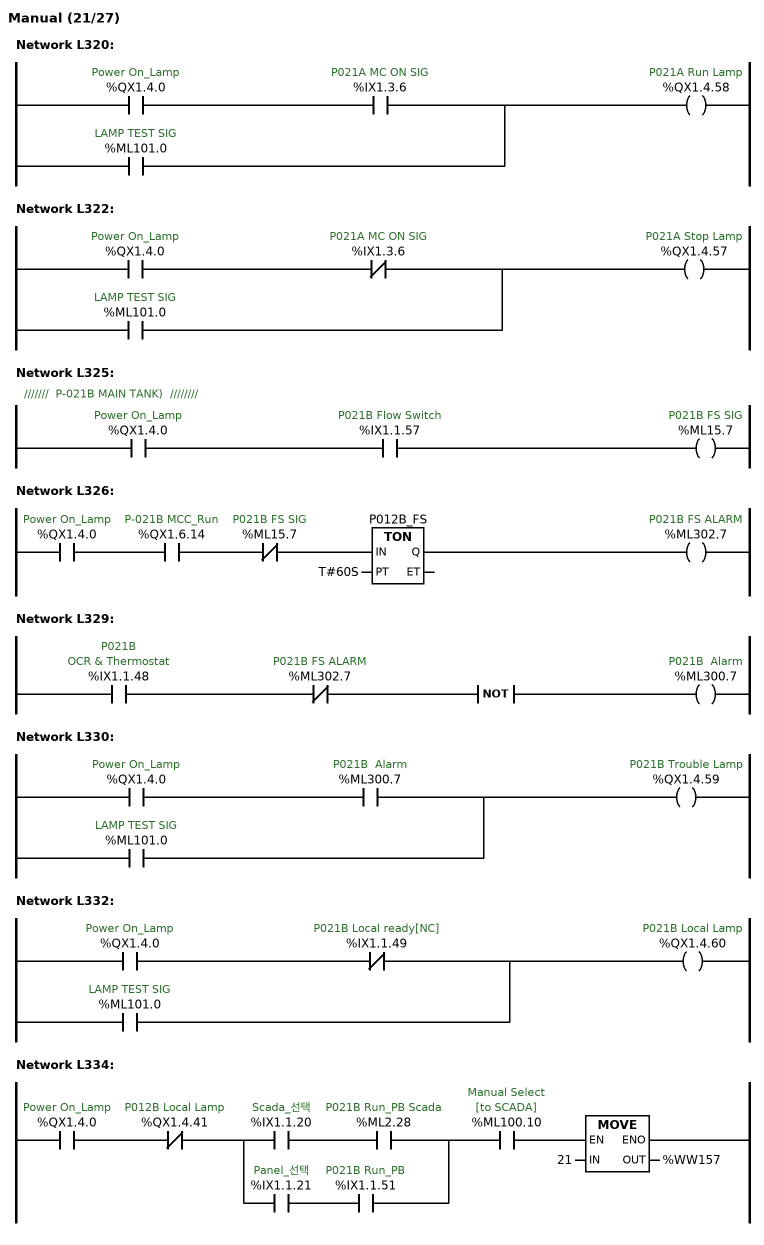
(* [picture p24: Manual rungs L320-L334] *)
(* Rung L320 *)
%QX1.4.58 := (%QX1.4.0 AND %IX1.3.6) OR %ML101.0;
(* Rung L322 *)
%QX1.4.57 := (%QX1.4.0 AND NOT %IX1.3.6) OR %ML101.0;
(* ///////  P-021B MAIN TANK)  //////// *)
(* Rung L325 *)
%ML15.7 := %QX1.4.0 AND %IX1.1.57;
(* Rung L326 *)
P012B_FS(IN := %QX1.4.0 AND %QX1.6.14 AND NOT %ML15.7, PT := T#60S);
%ML302.7 := P012B_FS.Q;
(* Rung L329 *)
%ML300.7 := NOT (%IX1.1.48 AND NOT %ML302.7);
(* Rung L330 *)
%QX1.4.59 := (%QX1.4.0 AND %ML300.7) OR %ML101.0;
(* Rung L332 *)
%QX1.4.60 := (%QX1.4.0 AND NOT %IX1.1.49) OR %ML101.0;
(* Rung L334 *)
IF %QX1.4.0 AND NOT %QX1.4.41 AND ((%IX1.1.20 AND %ML2.28) OR (%IX1.1.21 AND %IX1.1.51)) AND %ML100.10 THEN
    %WW157 := 21;
END_IF;

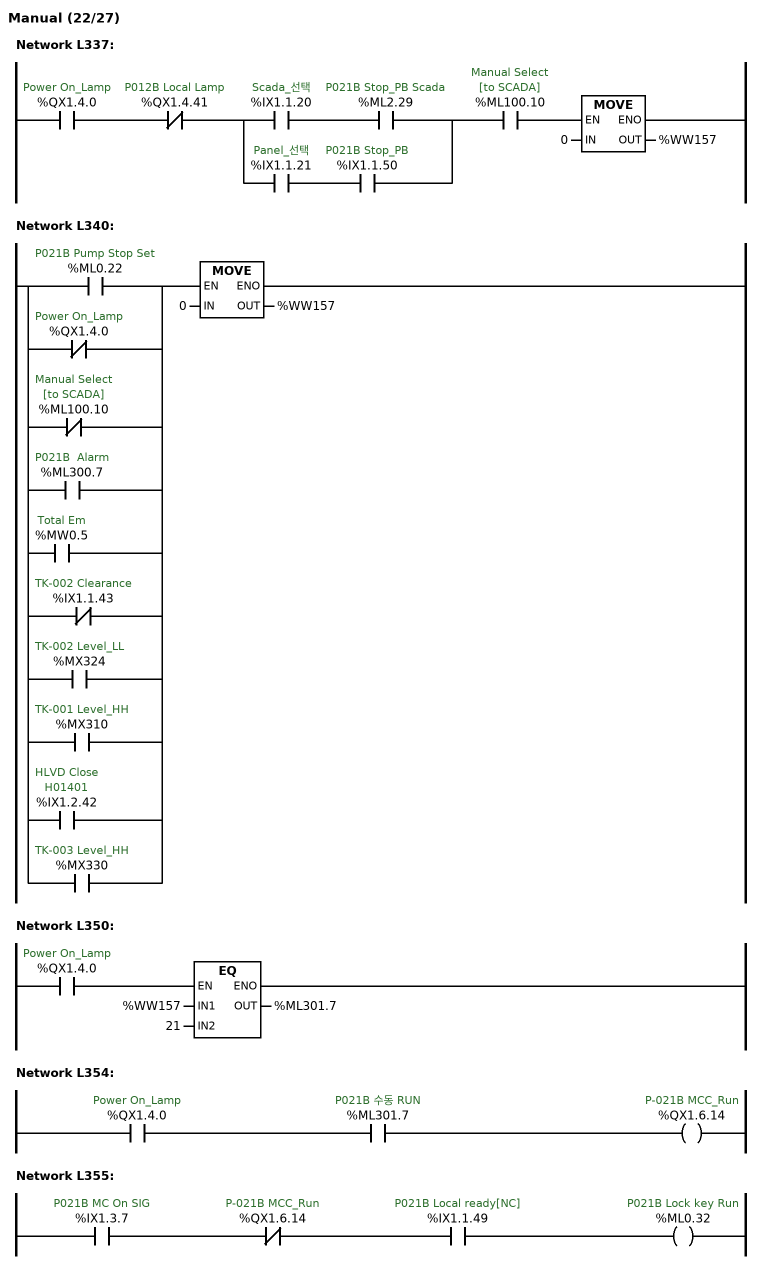
(* Rung L337 *)
IF %QX1.4.0 AND NOT %QX1.4.41 AND ((%IX1.1.20 AND %ML2.29) OR (%IX1.1.21 AND %IX1.1.50)) AND %ML100.10 THEN
    %WW157 := 0;
END_IF;
(* Rung L340 *)
IF %ML0.22 OR NOT %QX1.4.0 OR NOT %ML100.10 OR %ML300.7 OR %MW0.5 OR NOT %IX1.1.43 OR %MX324 OR %MX310 OR %IX1.2.42 OR %MX330 THEN
    %WW157 := 0;
END_IF;
(* Rung L350 *)
IF %QX1.4.0 THEN %ML301.7 := %WW157 = 21; END_IF;
(* Rung L354 *)
%QX1.6.14 := %QX1.4.0 AND %ML301.7;
(* Rung L355 *)
%ML0.32 := %IX1.3.7 AND NOT %QX1.6.14 AND %IX1.1.49;

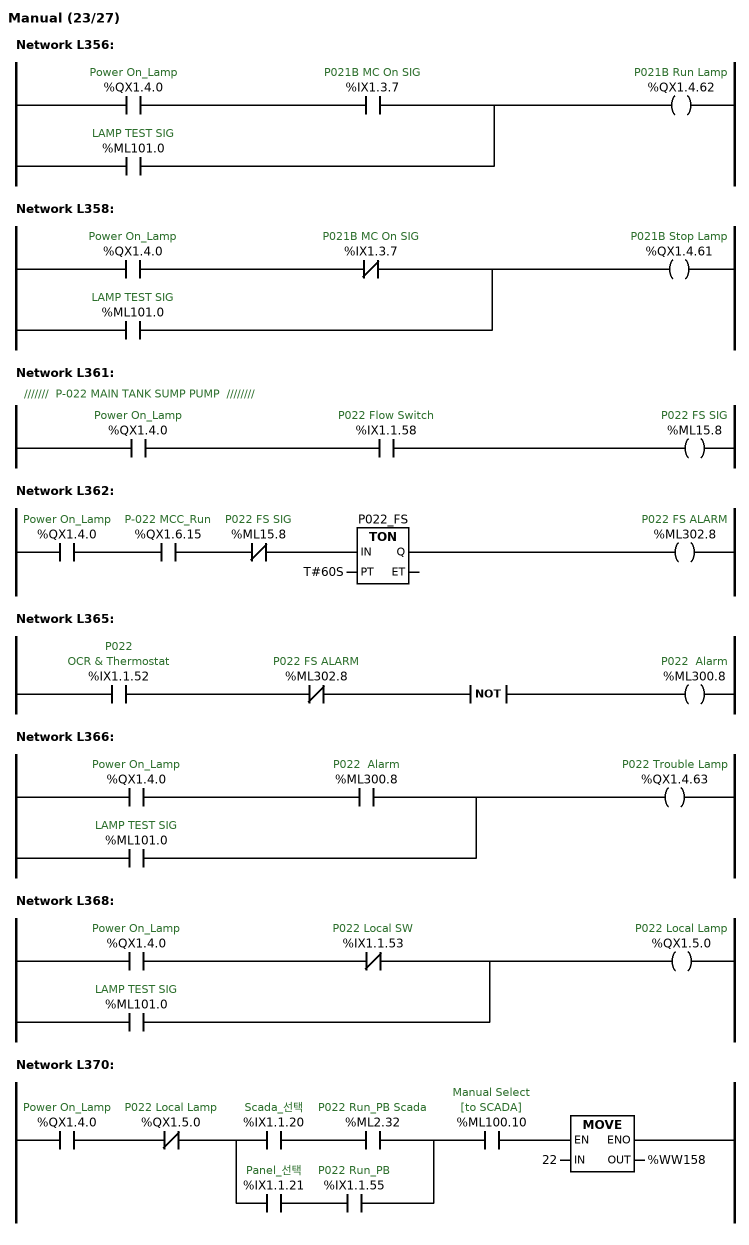
(* Rung L356 *)
%QX1.4.62 := (%QX1.4.0 AND %IX1.3.7) OR %ML101.0;
(* Rung L358 *)
%QX1.4.61 := (%QX1.4.0 AND NOT %IX1.3.7) OR %ML101.0;
(* ///////  P-022 MAIN TANK SUMP PUMP  //////// *)
(* Rung L361 *)
%ML15.8 := %QX1.4.0 AND %IX1.1.58;
(* Rung L362 *)
P022_FS(IN := %QX1.4.0 AND %QX1.6.15 AND NOT %ML15.8, PT := T#60S);
%ML302.8 := P022_FS.Q;
(* Rung L365 *)
%ML300.8 := NOT (%IX1.1.52 AND NOT %ML302.8);
(* Rung L366 *)
%QX1.4.63 := (%QX1.4.0 AND %ML300.8) OR %ML101.0;
(* Rung L368 *)
%QX1.5.0 := (%QX1.4.0 AND NOT %IX1.1.53) OR %ML101.0;
(* Rung L370 *)
IF %QX1.4.0 AND NOT %QX1.5.0 AND ((%IX1.1.20 AND %ML2.32) OR (%IX1.1.21 AND %IX1.1.55)) AND %ML100.10 THEN
    %WW158 := 22;
END_IF;

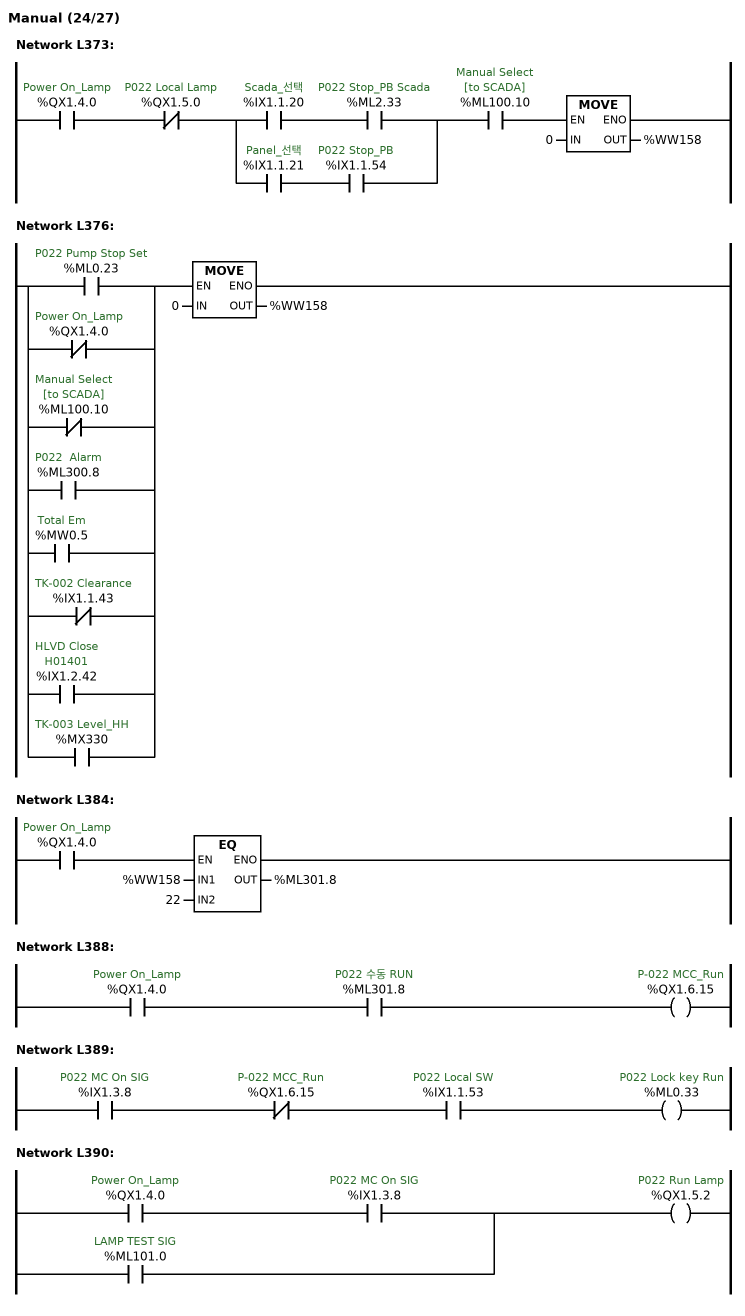
(* Rung L373 *)
IF %QX1.4.0 AND NOT %QX1.5.0 AND ((%IX1.1.20 AND %ML2.33) OR (%IX1.1.21 AND %IX1.1.54)) AND %ML100.10 THEN
    %WW158 := 0;
END_IF;
(* Rung L376 *)
IF %ML0.23 OR NOT %QX1.4.0 OR NOT %ML100.10 OR %ML300.8 OR %MW0.5 OR NOT %IX1.1.43 OR %IX1.2.42 OR %MX330 THEN
    %WW158 := 0;
END_IF;
(* Rung L384 *)
IF %QX1.4.0 THEN %ML301.8 := %WW158 = 22; END_IF;
(* Rung L388 *)
%QX1.6.15 := %QX1.4.0 AND %ML301.8;
(* Rung L389 *)
%ML0.33 := %IX1.3.8 AND NOT %QX1.6.15 AND %IX1.1.53;
(* Rung L390 *)
%QX1.5.2 := (%QX1.4.0 AND %IX1.3.8) OR %ML101.0;

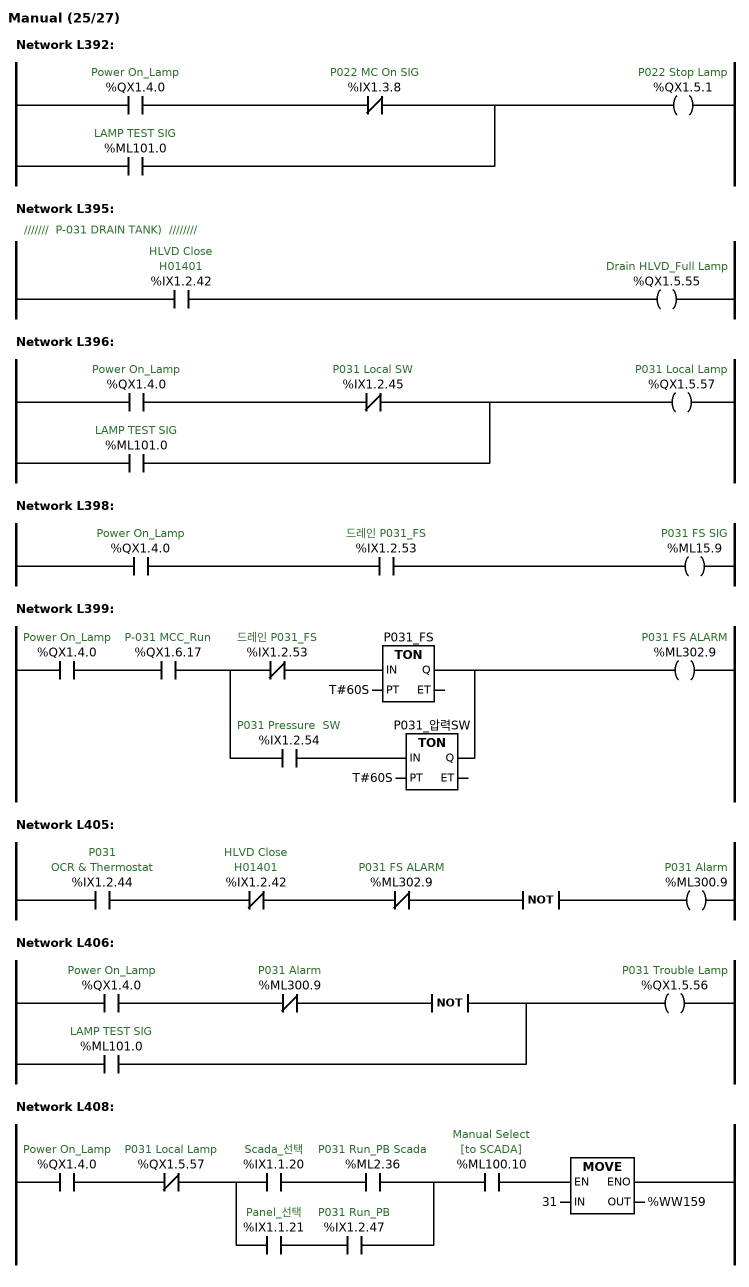
(* Rung L392 *)
%QX1.5.1 := (%QX1.4.0 AND NOT %IX1.3.8) OR %ML101.0;
(* ///////  P-031 DRAIN TANK)  //////// *)
(* Rung L395 *)
%QX1.5.55 := %IX1.2.42;
(* Rung L396 *)
%QX1.5.57 := (%QX1.4.0 AND NOT %IX1.2.45) OR %ML101.0;
(* Rung L398 *)
%ML15.9 := %QX1.4.0 AND %IX1.2.53;
(* Rung L399 *)
P031_FS(IN := %QX1.4.0 AND %QX1.6.17 AND NOT %IX1.2.53, PT := T#60S);
P031_압력SW(IN := %QX1.4.0 AND %QX1.6.17 AND %IX1.2.54, PT := T#60S);
%ML302.9 := P031_FS.Q OR P031_압력SW.Q;
(* Rung L405 *)
%ML300.9 := NOT (%IX1.2.44 AND NOT %IX1.2.42 AND NOT %ML302.9);
(* Rung L406 *)
%QX1.5.56 := NOT (%QX1.4.0 AND NOT %ML300.9) OR %ML101.0;
(* Rung L408 *)
IF %QX1.4.0 AND NOT %QX1.5.57 AND ((%IX1.1.20 AND %ML2.36) OR (%IX1.1.21 AND %IX1.2.47)) AND %ML100.10 THEN
    %WW159 := 31;
END_IF;

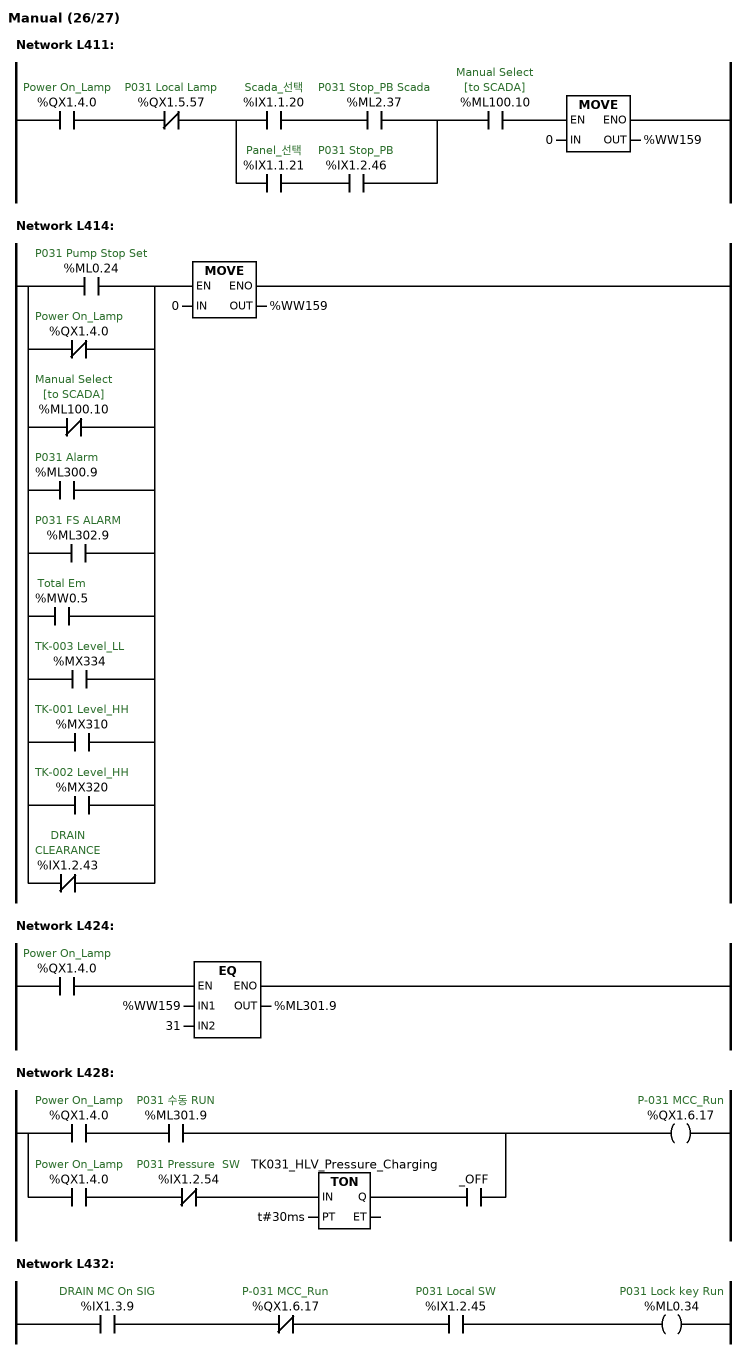
(* Rung L411 *)
IF %QX1.4.0 AND NOT %QX1.5.57 AND ((%IX1.1.20 AND %ML2.37) OR (%IX1.1.21 AND %IX1.2.46)) AND %ML100.10 THEN
    %WW159 := 0;
END_IF;
(* Rung L414 *)
IF %ML0.24 OR NOT %QX1.4.0 OR NOT %ML100.10 OR %ML300.9 OR %ML302.9 OR %MW0.5 OR %MX334 OR %MX310 OR %MX320 OR NOT %IX1.2.43 THEN
    %WW159 := 0;
END_IF;
(* Rung L424 *)
IF %QX1.4.0 THEN %ML301.9 := %WW159 = 31; END_IF;
(* Rung L428 *)
TK031_HLV_Pressure_Charging(IN := %QX1.4.0 AND NOT %IX1.2.54, PT := t#30ms);
%QX1.6.17 := (%QX1.4.0 AND %ML301.9) OR (TK031_HLV_Pressure_Charging.Q AND _OFF);
(* Rung L432 *)
%ML0.34 := %IX1.3.9 AND NOT %QX1.6.17 AND %IX1.2.45;

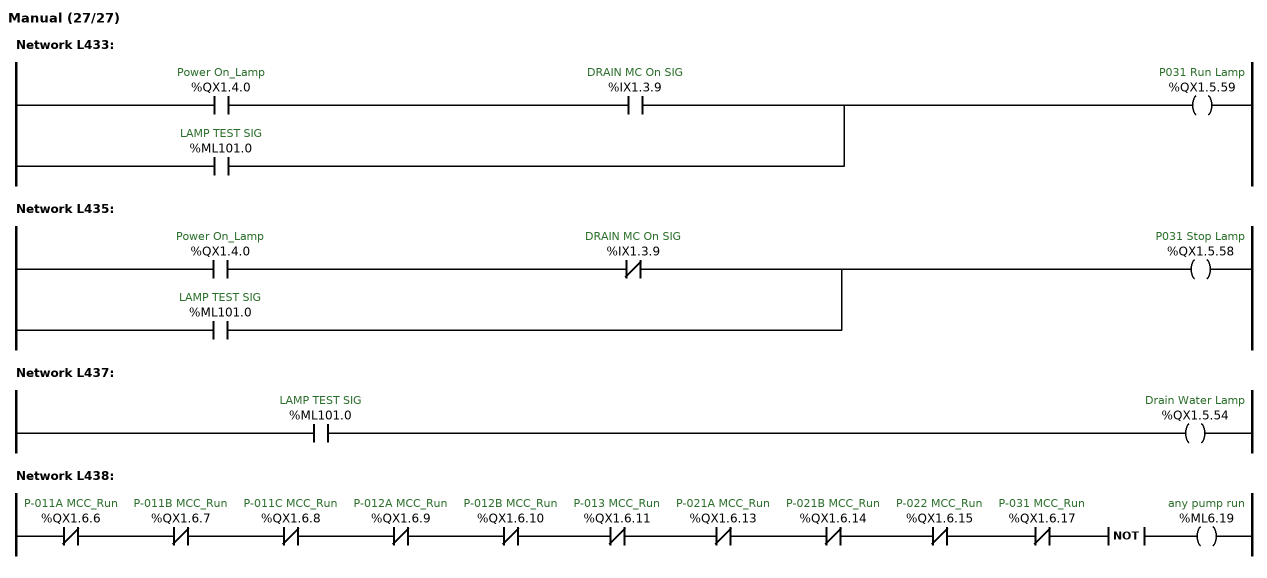
(* Rung L433 *)
%QX1.5.59 := (%QX1.4.0 AND %IX1.3.9) OR %ML101.0;
(* Rung L435 *)
%QX1.5.58 := (%QX1.4.0 AND NOT %IX1.3.9) OR %ML101.0;
(* Rung L437 *)
%QX1.5.54 := %ML101.0;
(* Rung L438 *)
%ML6.19 := NOT (NOT %QX1.6.6 AND NOT %QX1.6.7 AND NOT %QX1.6.8 AND NOT %QX1.6.9 AND NOT %QX1.6.10 AND NOT %QX1.6.11 AND NOT %QX1.6.13 AND NOT %QX1.6.14 AND NOT %QX1.6.15 AND NOT %QX1.6.17);
END_PROGRAM

PROGRAM Automatic (* task: 스캔 프로그램 *)
VAR
    AUTO_S_FS : TON;
END_VAR

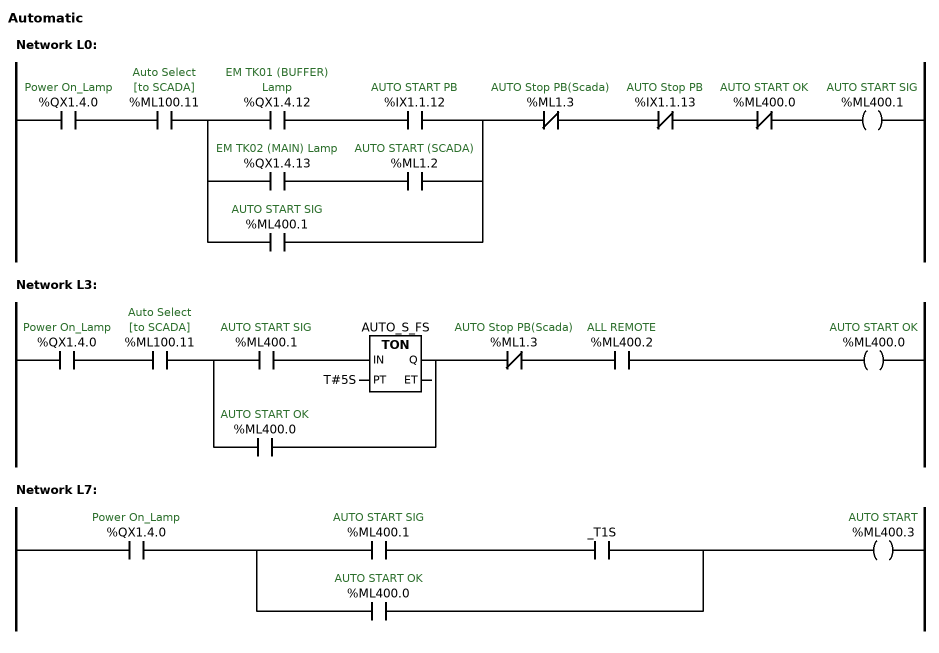
(* Rung L0 *)
%ML400.1 := %QX1.4.0 AND %ML100.11 AND ((%QX1.4.12 AND %IX1.1.12) OR (%QX1.4.13 AND %ML1.2) OR %ML400.1) AND NOT %ML1.3 AND NOT %IX1.1.13 AND NOT %ML400.0;
(* Rung L3 *)
AUTO_S_FS(IN := %QX1.4.0 AND %ML100.11 AND %ML400.1, PT := T#5S);
%ML400.0 := (AUTO_S_FS.Q OR (%QX1.4.0 AND %ML100.11 AND %ML400.0)) AND NOT %ML1.3 AND %ML400.2;
(* Rung L7 *)
%ML400.3 := %QX1.4.0 AND ((%ML400.1 AND _T1S) OR %ML400.0);
END_PROGRAM

PROGRAM Analog (* task: 스캔 프로그램 *)
VAR_EXTERNAL
    _0100_CH0_ACT : BOOL; (* AT %UX1.0.16 *) (* 아날로그입력 모듈: 채널0 운전중 *)
    _0100_CH0_DATA : INT; (* AT %UW1.0.2 *) (* 아날로그입력 모듈: 채널0 변환값 *)
    _0100_CH0_IDD : BOOL; (* AT %UX1.0.160 *) (* 아날로그입력 모듈: 채널0 입력단선검출 *)
    _0100_CH1_ACT : BOOL; (* AT %UX1.0.17 *) (* 아날로그입력 모듈: 채널1 운전중 *)
    _0100_CH1_DATA : INT; (* AT %UW1.0.3 *) (* 아날로그입력 모듈: 채널1 변환값 *)
    _0100_CH1_IDD : BOOL; (* AT %UX1.0.161 *) (* 아날로그입력 모듈: 채널1 입력단선검출 *)
    _0100_CH2_ACT : BOOL; (* AT %UX1.0.18 *) (* 아날로그입력 모듈: 채널2 운전중 *)
    _0100_CH2_DATA : INT; (* AT %UW1.0.4 *) (* 아날로그입력 모듈: 채널2 변환값 *)
    _0100_CH2_IDD : BOOL; (* AT %UX1.0.162 *) (* 아날로그입력 모듈: 채널2 입력단선검출 *)
    _0100_CH3_ACT : BOOL; (* AT %UX1.0.19 *) (* 아날로그입력 모듈: 채널3 운전중 *)
    _0100_CH3_DATA : INT; (* AT %UW1.0.5 *) (* 아날로그입력 모듈: 채널3 변환값 *)
    _0100_CH3_IDD : BOOL; (* AT %UX1.0.163 *) (* 아날로그입력 모듈: 채널3 입력단선검출 *)
    _0100_CH4_ACT : BOOL; (* AT %UX1.0.20 *) (* 아날로그입력 모듈: 채널4 운전중 *)
    _0100_CH4_DATA : INT; (* AT %UW1.0.6 *) (* 아날로그입력 모듈: 채널4 변환값 *)
    _0100_CH4_IDD : BOOL; (* AT %UX1.0.164 *) (* 아날로그입력 모듈: 채널4 입력단선검출 *)
    _0100_CH5_ACT : BOOL; (* AT %UX1.0.21 *) (* 아날로그입력 모듈: 채널5 운전중 *)
    _0100_CH5_DATA : INT; (* AT %UW1.0.7 *) (* 아날로그입력 모듈: 채널5 변환값 *)
    _0100_CH5_IDD : BOOL; (* AT %UX1.0.165 *) (* 아날로그입력 모듈: 채널5 입력단선검출 *)
    _0100_CH6_ACT : BOOL; (* AT %UX1.0.22 *) (* 아날로그입력 모듈: 채널6 운전중 *)
    _0100_CH6_DATA : INT; (* AT %UW1.0.8 *) (* 아날로그입력 모듈: 채널6 변환값 *)
    _0100_CH6_IDD : BOOL; (* AT %UX1.0.166 *) (* 아날로그입력 모듈: 채널6 입력단선검출 *)
    _0100_CH7_ACT : BOOL; (* AT %UX1.0.23 *) (* 아날로그입력 모듈: 채널7 운전중 *)
    _0100_CH7_DATA : INT; (* AT %UW1.0.9 *) (* 아날로그입력 모듈: 채널7 변환값 *)
    _0100_CH7_IDD : BOOL; (* AT %UX1.0.167 *) (* 아날로그입력 모듈: 채널7 입력단선검출 *)
END_VAR
VAR
    _t1 : BOOL;
    _t2 : BOOL;
    _t3 : BOOL;
    _t4 : BOOL;
END_VAR

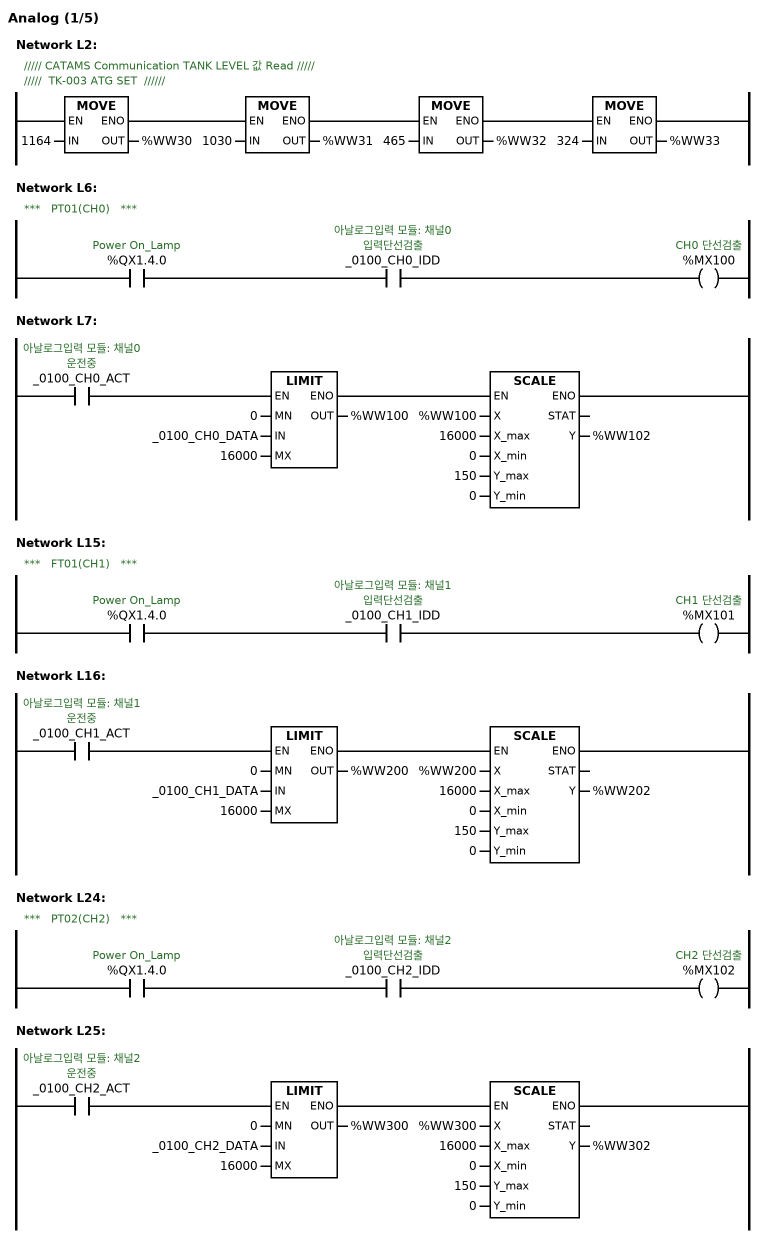
(* ///// CATAMS Communication TANK LEVEL 값 Read ///// *)
(* /////  TK-003 ATG SET  ////// *)
(* Rung L2 *)
%WW30 := 1164;
%WW31 := 1030;
%WW32 := 465;
%WW33 := 324;
(* ***   PT01(CH0)   *** *)
(* Rung L6 *)
%MX100 := %QX1.4.0 AND _0100_CH0_IDD;
(* Rung L7 *)
IF _0100_CH0_ACT THEN
    %WW100 := LIMIT(MN := 0, IN := _0100_CH0_DATA, MX := 16000);
    SCALE(X := %WW100, X_max := 16000, X_min := 0, Y_max := 150, Y_min := 0, Y => %WW102);
END_IF;
(* ***   FT01(CH1)   *** *)
(* Rung L15 *)
%MX101 := %QX1.4.0 AND _0100_CH1_IDD;
(* Rung L16 *)
IF _0100_CH1_ACT THEN
    %WW200 := LIMIT(MN := 0, IN := _0100_CH1_DATA, MX := 16000);
    SCALE(X := %WW200, X_max := 16000, X_min := 0, Y_max := 150, Y_min := 0, Y => %WW202);
END_IF;
(* ***   PT02(CH2)   *** *)
(* Rung L24 *)
%MX102 := %QX1.4.0 AND _0100_CH2_IDD;
(* Rung L25 *)
IF _0100_CH2_ACT THEN
    %WW300 := LIMIT(MN := 0, IN := _0100_CH2_DATA, MX := 16000);
    SCALE(X := %WW300, X_max := 16000, X_min := 0, Y_max := 150, Y_min := 0, Y => %WW302);
END_IF;

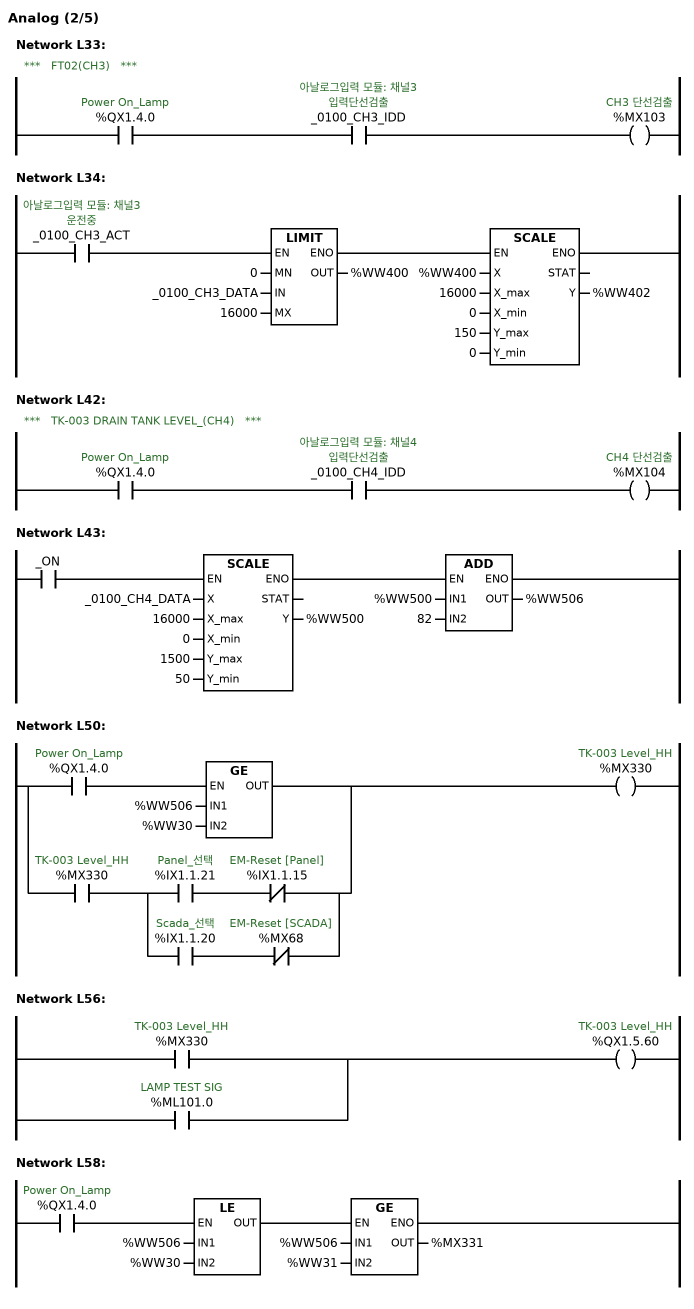
(* ***   FT02(CH3)   *** *)
(* Rung L33 *)
%MX103 := %QX1.4.0 AND _0100_CH3_IDD;
(* Rung L34 *)
IF _0100_CH3_ACT THEN
    %WW400 := LIMIT(MN := 0, IN := _0100_CH3_DATA, MX := 16000);
    SCALE(X := %WW400, X_max := 16000, X_min := 0, Y_max := 150, Y_min := 0, Y => %WW402);
END_IF;
(* ***   TK-003 DRAIN TANK LEVEL_(CH4)   *** *)
(* Rung L42 *)
%MX104 := %QX1.4.0 AND _0100_CH4_IDD;
(* Rung L43 *)
IF _ON THEN
    SCALE(X := _0100_CH4_DATA, X_max := 16000, X_min := 0, Y_max := 1500, Y_min := 50, Y => %WW500);
    %WW506 := %WW500 + 82;
END_IF;
(* Rung L50 *)
IF %QX1.4.0 THEN _t1 := %WW506 >= %WW30; END_IF;
%MX330 := _t1 OR (%MX330 AND ((%IX1.1.21 AND NOT %IX1.1.15) OR (%IX1.1.20 AND NOT %MX68)));
(* Rung L56 *)
%QX1.5.60 := %MX330 OR %ML101.0;
(* Rung L58 *)
IF %QX1.4.0 THEN _t2 := %WW506 <= %WW30; END_IF;
IF _t2 THEN %MX331 := %WW506 >= %WW31; END_IF;

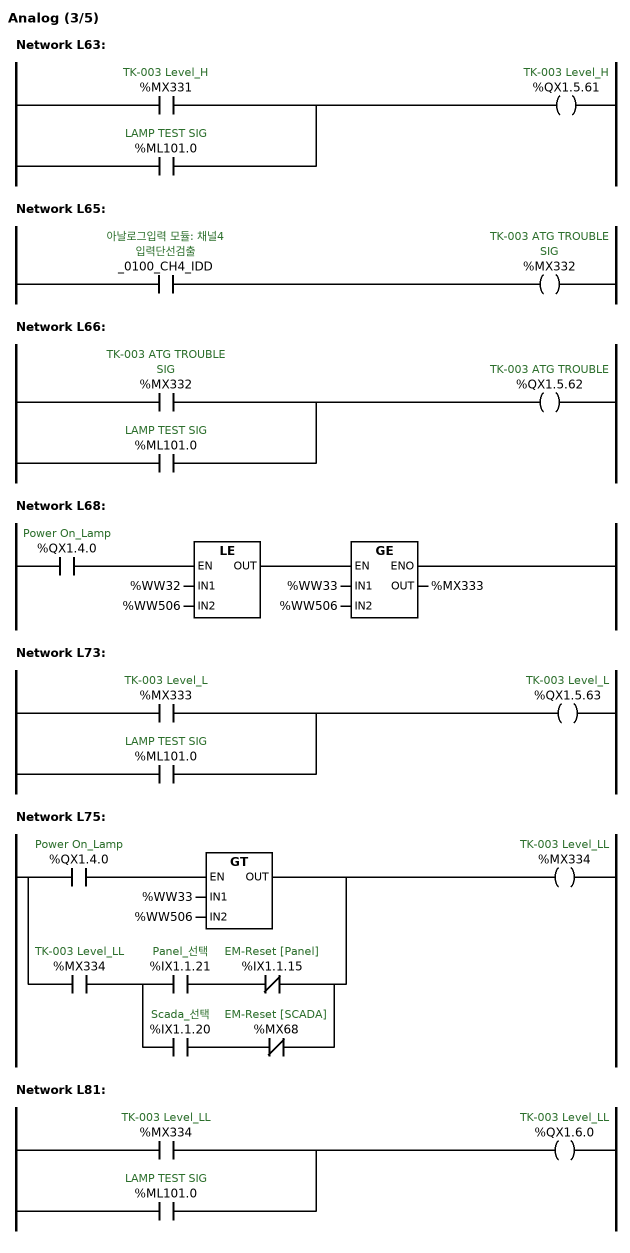
(* Rung L63 *)
%QX1.5.61 := %MX331 OR %ML101.0;
(* Rung L65 *)
%MX332 := _0100_CH4_IDD;
(* Rung L66 *)
%QX1.5.62 := %MX332 OR %ML101.0;
(* Rung L68 *)
IF %QX1.4.0 THEN _t3 := %WW32 <= %WW506; END_IF;
IF _t3 THEN %MX333 := %WW33 >= %WW506; END_IF;
(* Rung L73 *)
%QX1.5.63 := %MX333 OR %ML101.0;
(* Rung L75 *)
IF %QX1.4.0 THEN _t4 := %WW33 > %WW506; END_IF;
%MX334 := _t4 OR (%MX334 AND ((%IX1.1.21 AND NOT %IX1.1.15) OR (%IX1.1.20 AND NOT %MX68)));
(* Rung L81 *)
%QX1.6.0 := %MX334 OR %ML101.0;

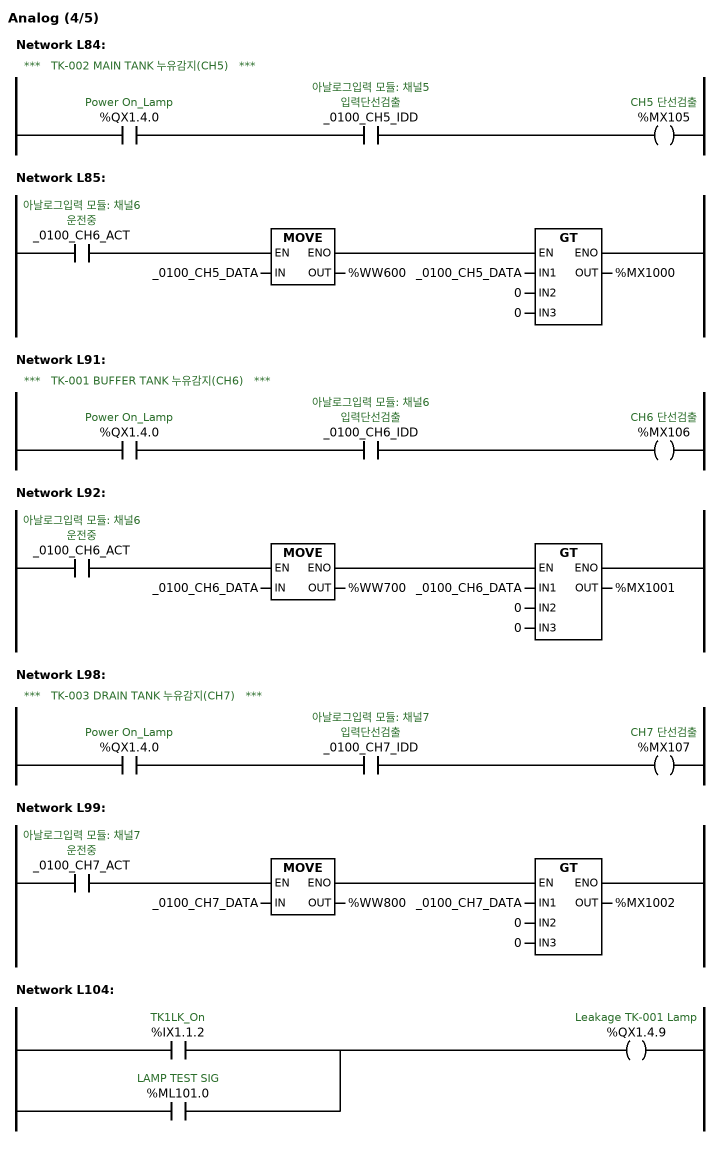
(* ***   TK-002 MAIN TANK 누유감지(CH5)   *** *)
(* Rung L84 *)
%MX105 := %QX1.4.0 AND _0100_CH5_IDD;
(* Rung L85 *)
IF _0100_CH6_ACT THEN
    %WW600 := _0100_CH5_DATA;
    %MX1000 := GT(_0100_CH5_DATA, 0, 0);
END_IF;
(* ***   TK-001 BUFFER TANK 누유감지(CH6)   *** *)
(* Rung L91 *)
%MX106 := %QX1.4.0 AND _0100_CH6_IDD;
(* Rung L92 *)
IF _0100_CH6_ACT THEN
    %WW700 := _0100_CH6_DATA;
    %MX1001 := GT(_0100_CH6_DATA, 0, 0);
END_IF;
(* ***   TK-003 DRAIN TANK 누유감지(CH7)   *** *)
(* Rung L98 *)
%MX107 := %QX1.4.0 AND _0100_CH7_IDD;
(* Rung L99 *)
IF _0100_CH7_ACT THEN
    %WW800 := _0100_CH7_DATA;
    %MX1002 := GT(_0100_CH7_DATA, 0, 0);
END_IF;
(* Rung L104 *)
%QX1.4.9 := %IX1.1.2 OR %ML101.0;

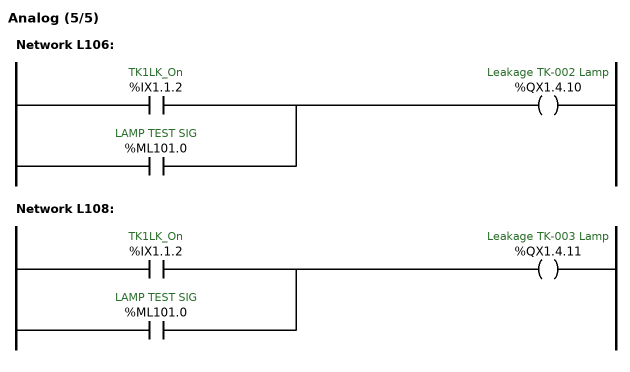
(* Rung L106 *)
%QX1.4.10 := %IX1.1.2 OR %ML101.0;
(* Rung L108 *)
%QX1.4.11 := %IX1.1.2 OR %ML101.0;
END_PROGRAM

PROGRAM Scada (* task: 스캔 프로그램 *)

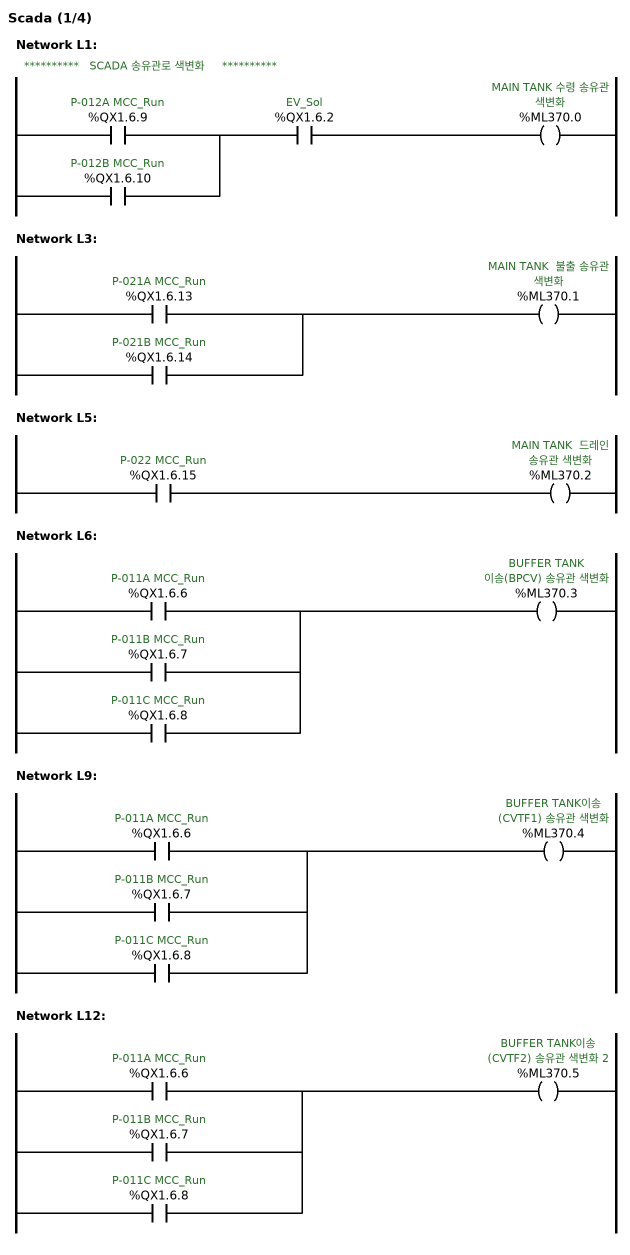
(* **********   SCADA 송유관로 색변화     ********** *)
(* Rung L1 *)
%ML370.0 := (%QX1.6.9 OR %QX1.6.10) AND %QX1.6.2;
(* Rung L3 *)
%ML370.1 := %QX1.6.13 OR %QX1.6.14;
(* Rung L5 *)
%ML370.2 := %QX1.6.15;
(* Rung L6 *)
%ML370.3 := %QX1.6.6 OR %QX1.6.7 OR %QX1.6.8;
(* Rung L9 *)
%ML370.4 := %QX1.6.6 OR %QX1.6.7 OR %QX1.6.8;
(* Rung L12 *)
%ML370.5 := %QX1.6.6 OR %QX1.6.7 OR %QX1.6.8;

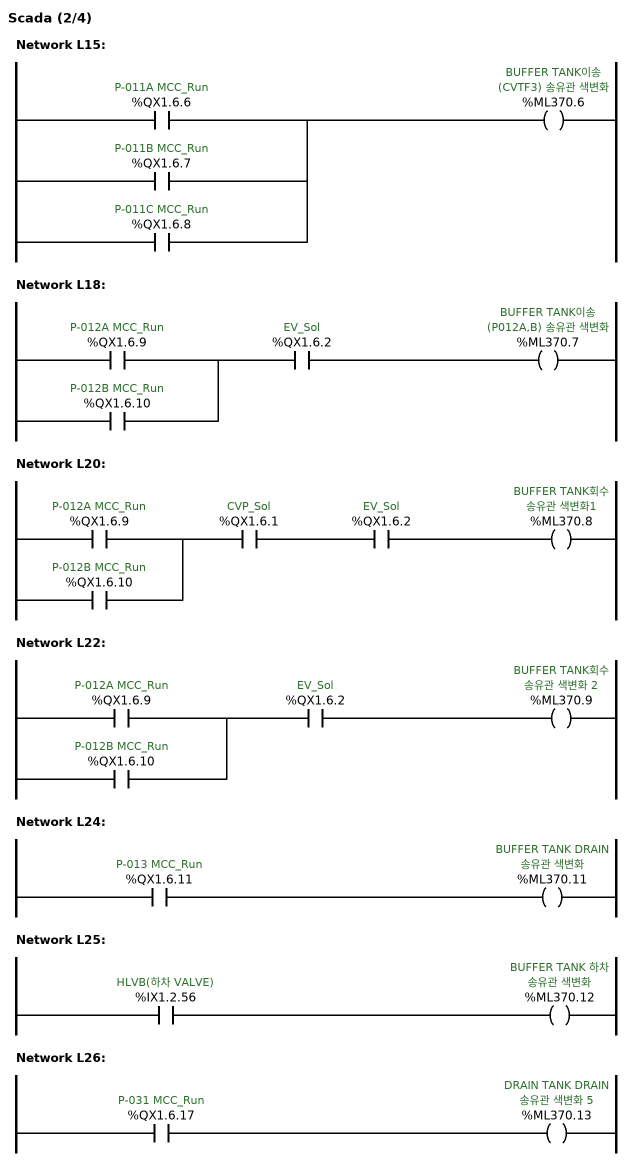
(* Rung L15 *)
%ML370.6 := %QX1.6.6 OR %QX1.6.7 OR %QX1.6.8;
(* Rung L18 *)
%ML370.7 := (%QX1.6.9 OR %QX1.6.10) AND %QX1.6.2;
(* Rung L20 *)
%ML370.8 := (%QX1.6.9 OR %QX1.6.10) AND %QX1.6.1 AND %QX1.6.2;
(* Rung L22 *)
%ML370.9 := (%QX1.6.9 OR %QX1.6.10) AND %QX1.6.2;
(* Rung L24 *)
%ML370.11 := %QX1.6.11;
(* Rung L25 *)
%ML370.12 := %IX1.2.56;
(* Rung L26 *)
%ML370.13 := %QX1.6.17;

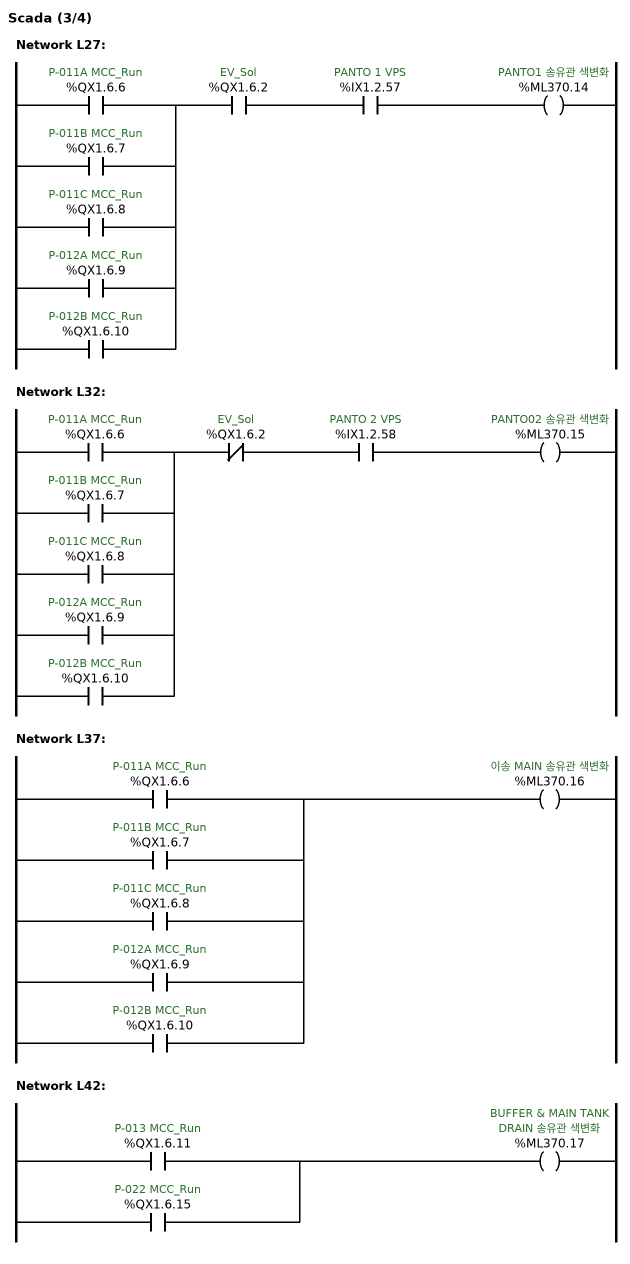
(* Rung L27 *)
%ML370.14 := (%QX1.6.6 OR %QX1.6.7 OR %QX1.6.8 OR %QX1.6.9 OR %QX1.6.10) AND %QX1.6.2 AND %IX1.2.57;
(* Rung L32 *)
%ML370.15 := (%QX1.6.6 OR %QX1.6.7 OR %QX1.6.8 OR %QX1.6.9 OR %QX1.6.10) AND NOT %QX1.6.2 AND %IX1.2.58;
(* Rung L37 *)
%ML370.16 := %QX1.6.6 OR %QX1.6.7 OR %QX1.6.8 OR %QX1.6.9 OR %QX1.6.10;
(* Rung L42 *)
%ML370.17 := %QX1.6.11 OR %QX1.6.15;

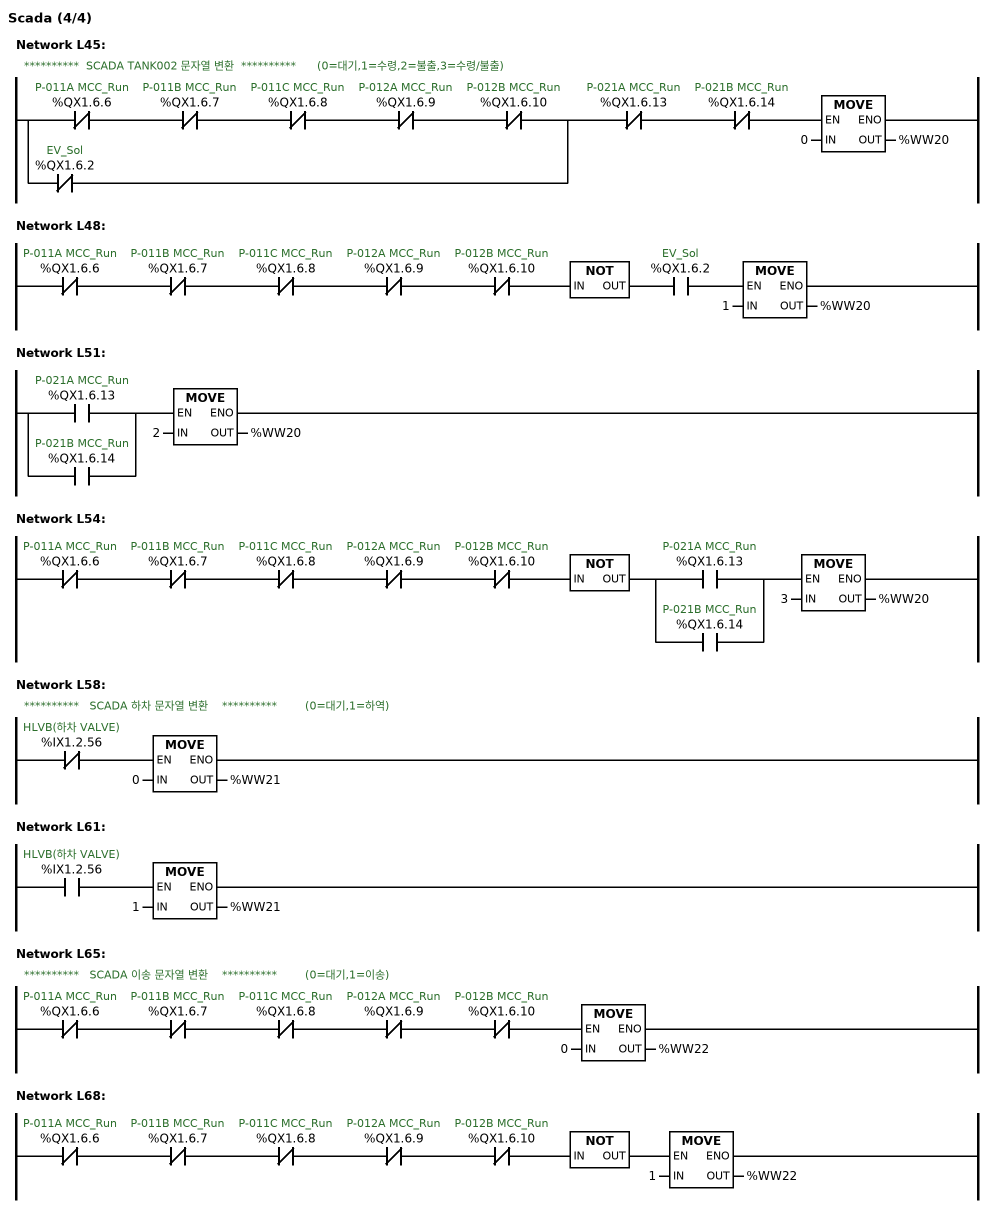
(* **********  SCADA TANK002 문자열 변환  **********      (0=대기,1=수령,2=불출,3=수령/불출) *)
(* Rung L45 *)
IF ((NOT %QX1.6.6 AND NOT %QX1.6.7 AND NOT %QX1.6.8 AND NOT %QX1.6.9 AND NOT %QX1.6.10) OR NOT %QX1.6.2) AND NOT %QX1.6.13 AND NOT %QX1.6.14 THEN
    %WW20 := 0;
END_IF;
(* Rung L48 *)
IF (NOT (NOT %QX1.6.6 AND NOT %QX1.6.7 AND NOT %QX1.6.8 AND NOT %QX1.6.9 AND NOT %QX1.6.10)) AND %QX1.6.2 THEN
    %WW20 := 1;
END_IF;
(* Rung L51 *)
IF %QX1.6.13 OR %QX1.6.14 THEN %WW20 := 2; END_IF;
(* Rung L54 *)
IF (NOT (NOT %QX1.6.6 AND NOT %QX1.6.7 AND NOT %QX1.6.8 AND NOT %QX1.6.9 AND NOT %QX1.6.10)) AND (%QX1.6.13 OR %QX1.6.14) THEN
    %WW20 := 3;
END_IF;
(* **********   SCADA 하차 문자열 변환    **********        (0=대기,1=하역) *)
(* Rung L58 *)
IF NOT %IX1.2.56 THEN %WW21 := 0; END_IF;
(* Rung L61 *)
IF %IX1.2.56 THEN %WW21 := 1; END_IF;
(* **********   SCADA 이송 문자열 변환    **********        (0=대기,1=이송) *)
(* Rung L65 *)
IF NOT %QX1.6.6 AND NOT %QX1.6.7 AND NOT %QX1.6.8 AND NOT %QX1.6.9 AND NOT %QX1.6.10 THEN
    %WW22 := 0;
END_IF;
(* Rung L68 *)
IF NOT (NOT %QX1.6.6 AND NOT %QX1.6.7 AND NOT %QX1.6.8 AND NOT %QX1.6.9 AND NOT %QX1.6.10) THEN
    %WW22 := 1;
END_IF;
END_PROGRAM

PROGRAM Communication (* task: 스캔 프로그램 *)
VAR
    TK001_TROUBLE : TON; (* TK_001_TROUBLE DELAY TIMER *)
    TK002_TROUBLE : TON; (* TK_001_TROUBLE DELAY TIMER *)
END_VAR
VAR_EXTERNAL
    _0100_CH4_DATA : INT; (* AT %UW1.0.6 *) (* 아날로그입력 모듈: 채널4 변환값 *)
END_VAR
VAR
    _t1 : BOOL;
    _t2 : BOOL;
    _t3 : BOOL;
    _t4 : BOOL;
    _t5 : BOOL;
    _t6 : BOOL;
    _t7 : BOOL;
    _t8 : BOOL;
    _t9 : BOOL;
    _t10 : BOOL;
END_VAR

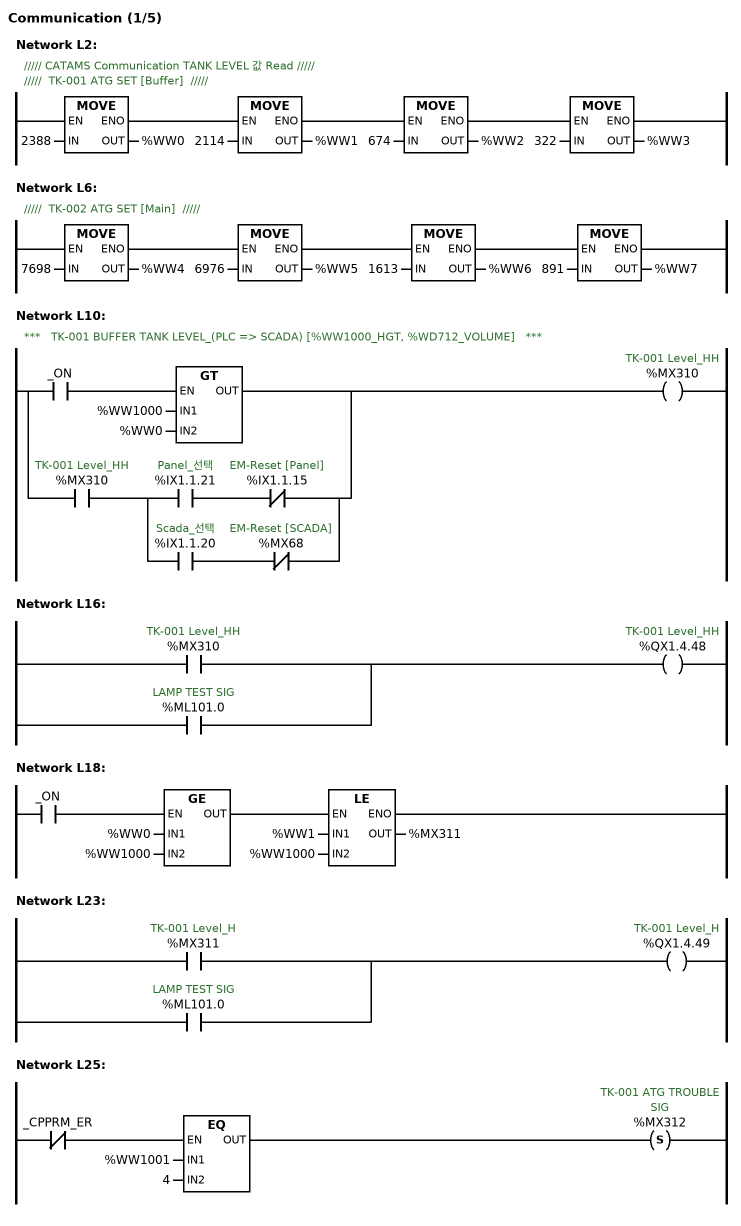
(* ///// CATAMS Communication TANK LEVEL 값 Read ///// *)
(* /////  TK-001 ATG SET [Buffer]  ///// *)
(* Rung L2 *)
%WW0 := 2388;
%WW1 := 2114;
%WW2 := 674;
%WW3 := 322;
(* /////  TK-002 ATG SET [Main]  ///// *)
(* Rung L6 *)
%WW4 := 7698;
%WW5 := 6976;
%WW6 := 1613;
%WW7 := 891;
(* ***   TK-001 BUFFER TANK LEVEL_(PLC => SCADA) [%WW1000_HGT, %WD712_VOLUME]   *** *)
(* Rung L10 *)
IF _ON THEN _t1 := %WW1000 > %WW0; END_IF;
%MX310 := _t1 OR (%MX310 AND ((%IX1.1.21 AND NOT %IX1.1.15) OR (%IX1.1.20 AND NOT %MX68)));
(* Rung L16 *)
%QX1.4.48 := %MX310 OR %ML101.0;
(* Rung L18 *)
IF _ON THEN _t2 := %WW0 >= %WW1000; END_IF;
IF _t2 THEN %MX311 := %WW1 <= %WW1000; END_IF;
(* Rung L23 *)
%QX1.4.49 := %MX311 OR %ML101.0;
(* Rung L25 *)
IF NOT _CPPRM_ER THEN _t3 := %WW1001 = 4; END_IF;
IF _t3 THEN %MX312 := TRUE; END_IF;

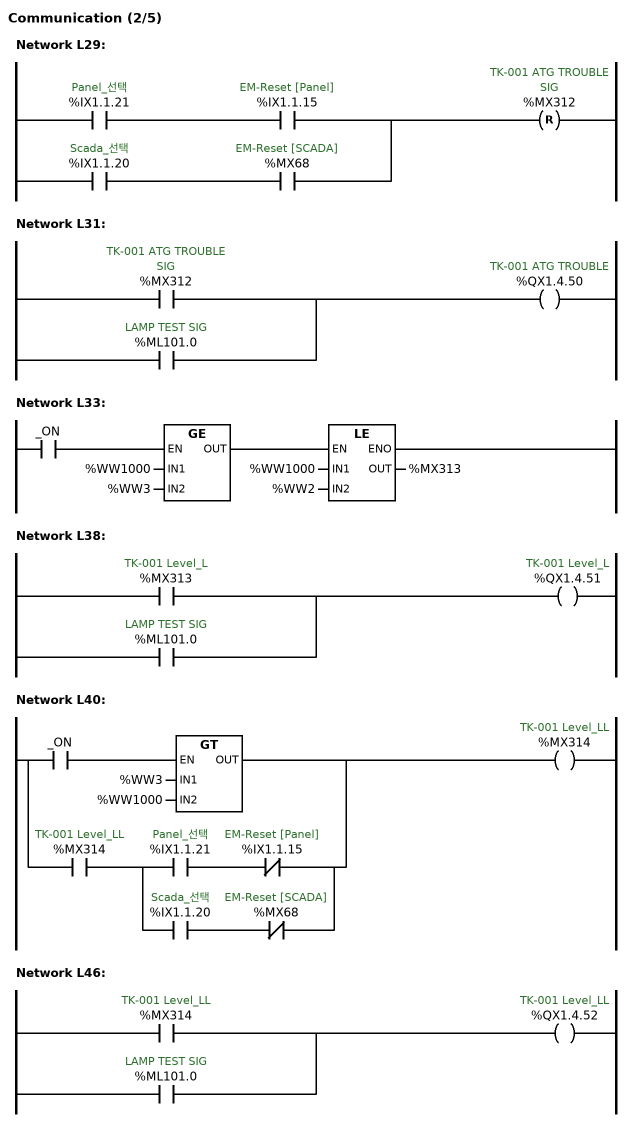
(* Rung L29 *)
IF (%IX1.1.21 AND %IX1.1.15) OR (%IX1.1.20 AND %MX68) THEN %MX312 := FALSE; END_IF;
(* Rung L31 *)
%QX1.4.50 := %MX312 OR %ML101.0;
(* Rung L33 *)
IF _ON THEN _t4 := %WW1000 >= %WW3; END_IF;
IF _t4 THEN %MX313 := %WW1000 <= %WW2; END_IF;
(* Rung L38 *)
%QX1.4.51 := %MX313 OR %ML101.0;
(* Rung L40 *)
IF _ON THEN _t5 := %WW3 > %WW1000; END_IF;
%MX314 := _t5 OR (%MX314 AND ((%IX1.1.21 AND NOT %IX1.1.15) OR (%IX1.1.20 AND NOT %MX68)));
(* Rung L46 *)
%QX1.4.52 := %MX314 OR %ML101.0;

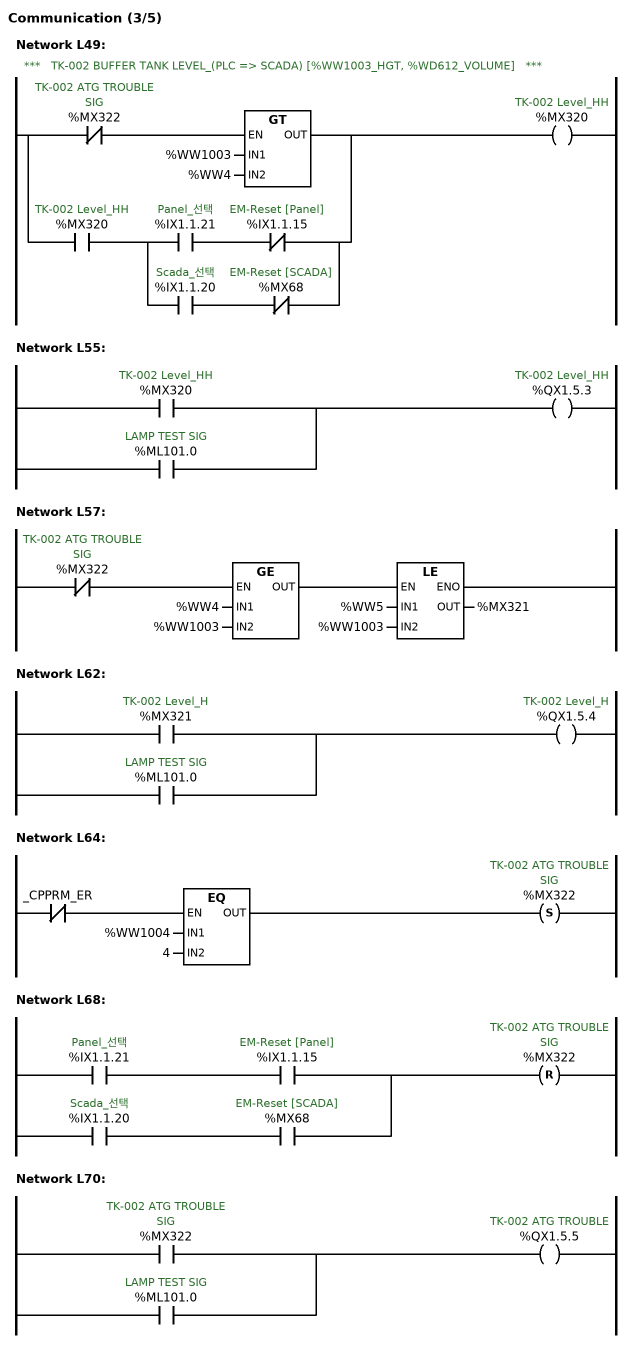
(* ***   TK-002 BUFFER TANK LEVEL_(PLC => SCADA) [%WW1003_HGT, %WD612_VOLUME]   *** *)
(* Rung L49 *)
IF NOT %MX322 THEN _t6 := %WW1003 > %WW4; END_IF;
%MX320 := _t6 OR (%MX320 AND ((%IX1.1.21 AND NOT %IX1.1.15) OR (%IX1.1.20 AND NOT %MX68)));
(* Rung L55 *)
%QX1.5.3 := %MX320 OR %ML101.0;
(* Rung L57 *)
IF NOT %MX322 THEN _t7 := %WW4 >= %WW1003; END_IF;
IF _t7 THEN %MX321 := %WW5 <= %WW1003; END_IF;
(* Rung L62 *)
%QX1.5.4 := %MX321 OR %ML101.0;
(* Rung L64 *)
IF NOT _CPPRM_ER THEN _t8 := %WW1004 = 4; END_IF;
IF _t8 THEN %MX322 := TRUE; END_IF;
(* Rung L68 *)
IF (%IX1.1.21 AND %IX1.1.15) OR (%IX1.1.20 AND %MX68) THEN %MX322 := FALSE; END_IF;
(* Rung L70 *)
%QX1.5.5 := %MX322 OR %ML101.0;

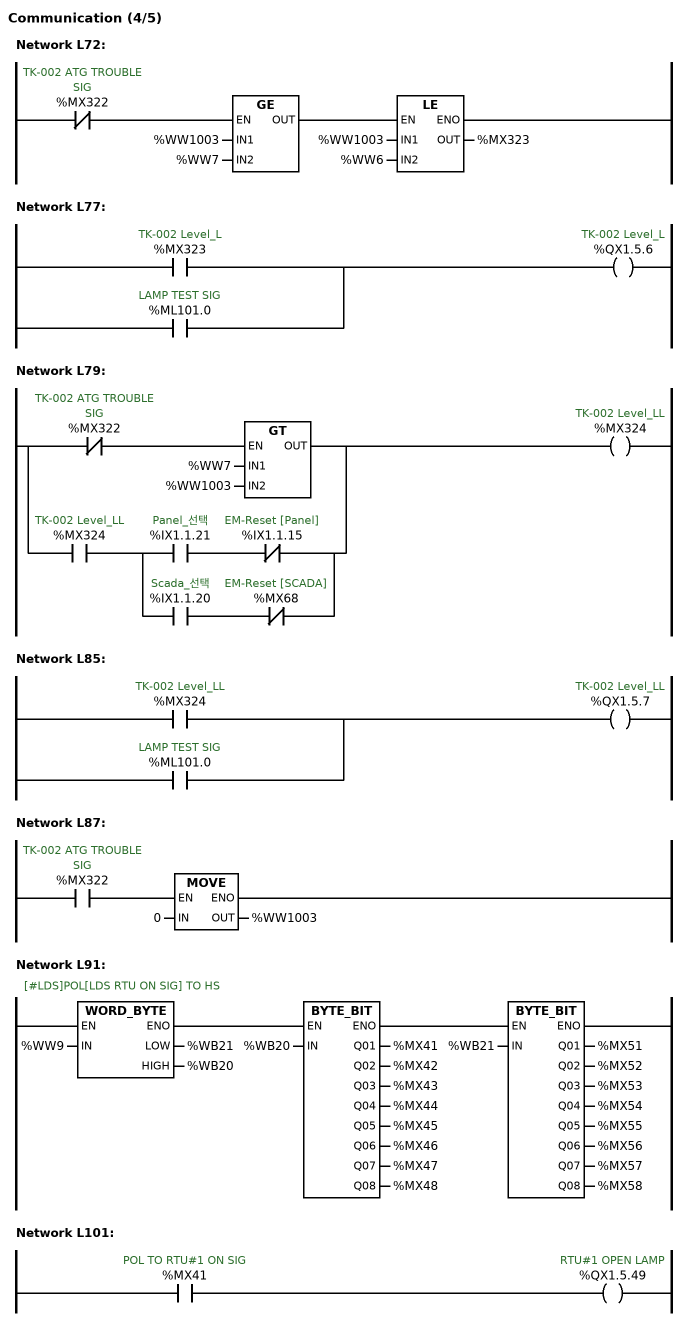
(* Rung L72 *)
IF NOT %MX322 THEN _t9 := %WW1003 >= %WW7; END_IF;
IF _t9 THEN %MX323 := %WW1003 <= %WW6; END_IF;
(* Rung L77 *)
%QX1.5.6 := %MX323 OR %ML101.0;
(* Rung L79 *)
IF NOT %MX322 THEN _t10 := %WW7 > %WW1003; END_IF;
%MX324 := _t10 OR (%MX324 AND ((%IX1.1.21 AND NOT %IX1.1.15) OR (%IX1.1.20 AND NOT %MX68)));
(* Rung L85 *)
%QX1.5.7 := %MX324 OR %ML101.0;
(* Rung L87 *)
IF %MX322 THEN %WW1003 := 0; END_IF;
(* [#LDS]POL[LDS RTU ON SIG] TO HS *)
(* Rung L91 *)
%WB21 := WORD_BYTE(IN := %WW9, HIGH => %WB20);
%MX41 := BYTE_BIT(IN := %WB20, Q02 => %MX42, Q03 => %MX43, Q04 => %MX44, Q05 => %MX45, Q06 => %MX46, Q07 => %MX47, Q08 => %MX48);
%MX51 := BYTE_BIT(IN := %WB21, Q02 => %MX52, Q03 => %MX53, Q04 => %MX54, Q05 => %MX55, Q06 => %MX56, Q07 => %MX57, Q08 => %MX58);
(* Rung L101 *)
%QX1.5.49 := %MX41;

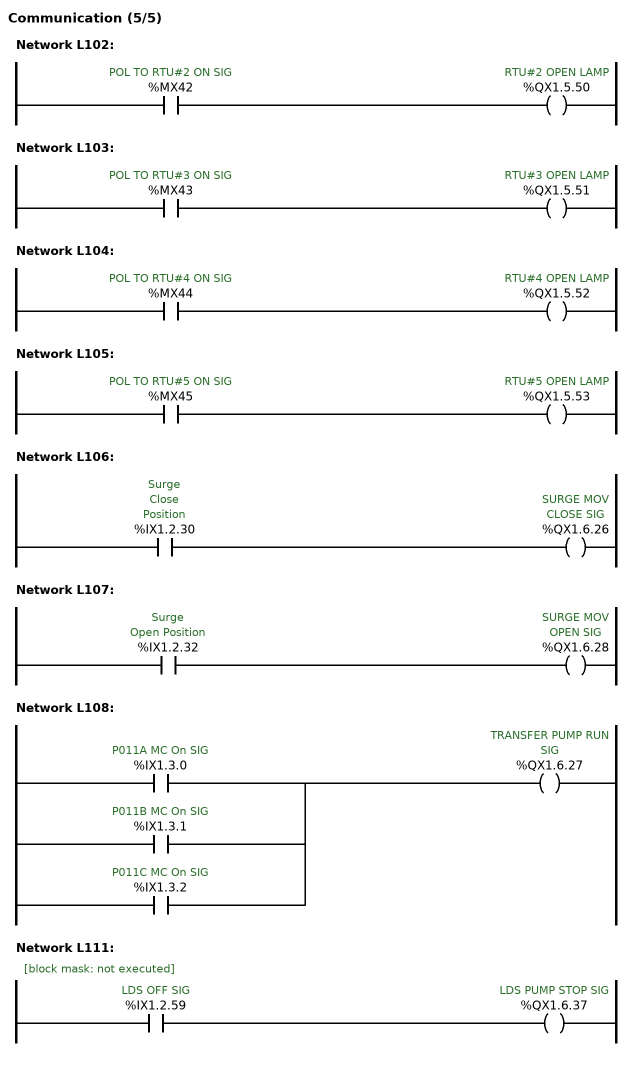
(* Rung L102 *)
%QX1.5.50 := %MX42;
(* Rung L103 *)
%QX1.5.51 := %MX43;
(* Rung L104 *)
%QX1.5.52 := %MX44;
(* Rung L105 *)
%QX1.5.53 := %MX45;
(* Rung L106 *)
%QX1.6.26 := %IX1.2.30;
(* Rung L107 *)
%QX1.6.28 := %IX1.2.32;
(* Rung L108 *)
%QX1.6.27 := %IX1.3.0 OR %IX1.3.1 OR %IX1.3.2;
(* Rung L111 is block-masked: not executed *)
// %QX1.6.37 := %IX1.2.59;
END_PROGRAM

PROGRAM Setting (* task: 스캔 프로그램 *)
VAR
    _e1 : R_TRIG;
    _e2 : R_TRIG;
    _e3 : R_TRIG;
    _e4 : R_TRIG;
    _e5 : R_TRIG;
    _e6 : R_TRIG;
    _e7 : R_TRIG;
    _e8 : R_TRIG;
    _e9 : R_TRIG;
    _t10 : BOOL;
    _t11 : BOOL;
    _t12 : BOOL;
    _t13 : BOOL;
    _t14 : BOOL;
    _t15 : BOOL;
    _t16 : BOOL;
    _t17 : BOOL;
    _t18 : BOOL;
    _t19 : BOOL;
    _t20 : BOOL;
    _t21 : BOOL;
    _t22 : BOOL;
    _t23 : BOOL;
END_VAR

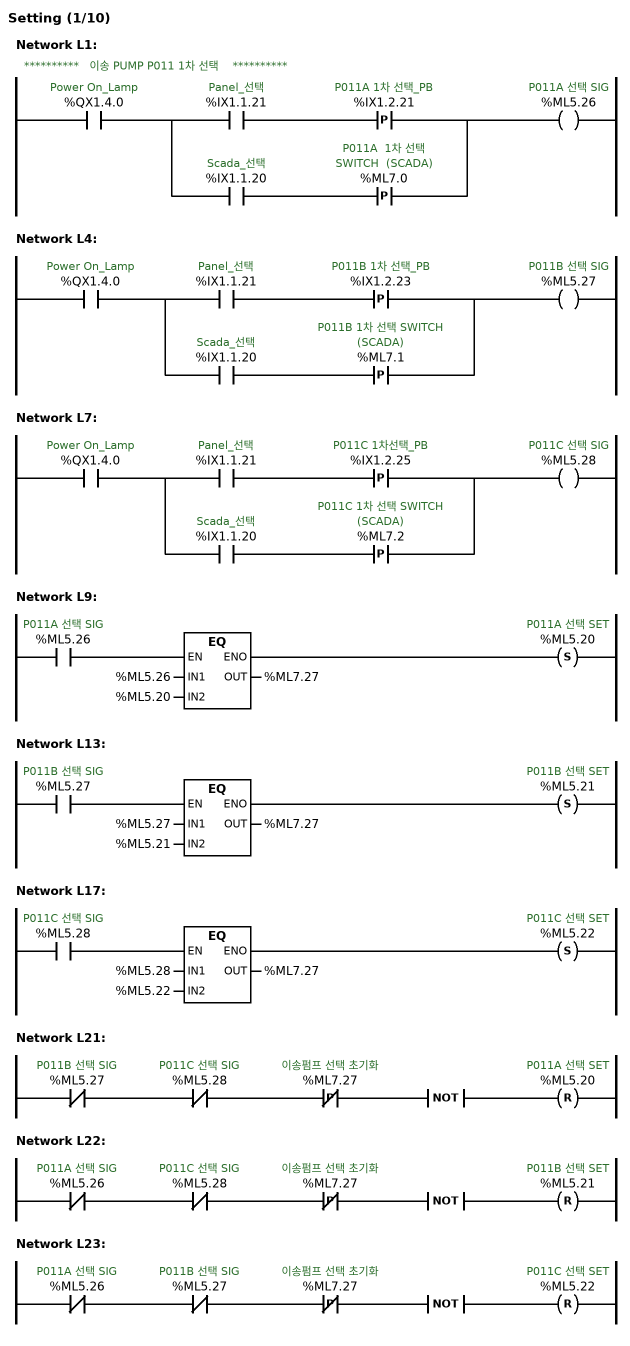
(* **********   이송 PUMP P011 1차 선택    ********** *)
(* Rung L1 *)
_e1(CLK := %IX1.2.21);
_e2(CLK := %ML7.0);
%ML5.26 := %QX1.4.0 AND ((%IX1.1.21 AND _e1.Q) OR (%IX1.1.20 AND _e2.Q));
(*  *)
(* Rung L4 *)
_e3(CLK := %IX1.2.23);
_e4(CLK := %ML7.1);
%ML5.27 := %QX1.4.0 AND ((%IX1.1.21 AND _e3.Q) OR (%IX1.1.20 AND _e4.Q));
(*  *)
(* Rung L7 *)
_e5(CLK := %IX1.2.25);
_e6(CLK := %ML7.2);
%ML5.28 := %QX1.4.0 AND ((%IX1.1.21 AND _e5.Q) OR (%IX1.1.20 AND _e6.Q));
(* Rung L9 *)
IF %ML5.26 THEN
    %ML7.27 := %ML5.26 = %ML5.20;
    %ML5.20 := TRUE;
END_IF;
(* Rung L13 *)
IF %ML5.27 THEN
    %ML7.27 := %ML5.27 = %ML5.21;
    %ML5.21 := TRUE;
END_IF;
(* Rung L17 *)
IF %ML5.28 THEN
    %ML7.27 := %ML5.28 = %ML5.22;
    %ML5.22 := TRUE;
END_IF;
(* Rung L21 *)
_e7(CLK := %ML7.27);
IF NOT (NOT %ML5.27 AND NOT %ML5.28 AND NOT _e7.Q) THEN %ML5.20 := FALSE; END_IF;
(* Rung L22 *)
_e8(CLK := %ML7.27);
IF NOT (NOT %ML5.26 AND NOT %ML5.28 AND NOT _e8.Q) THEN %ML5.21 := FALSE; END_IF;
(* Rung L23 *)
_e9(CLK := %ML7.27);
IF NOT (NOT %ML5.26 AND NOT %ML5.27 AND NOT _e9.Q) THEN %ML5.22 := FALSE; END_IF;

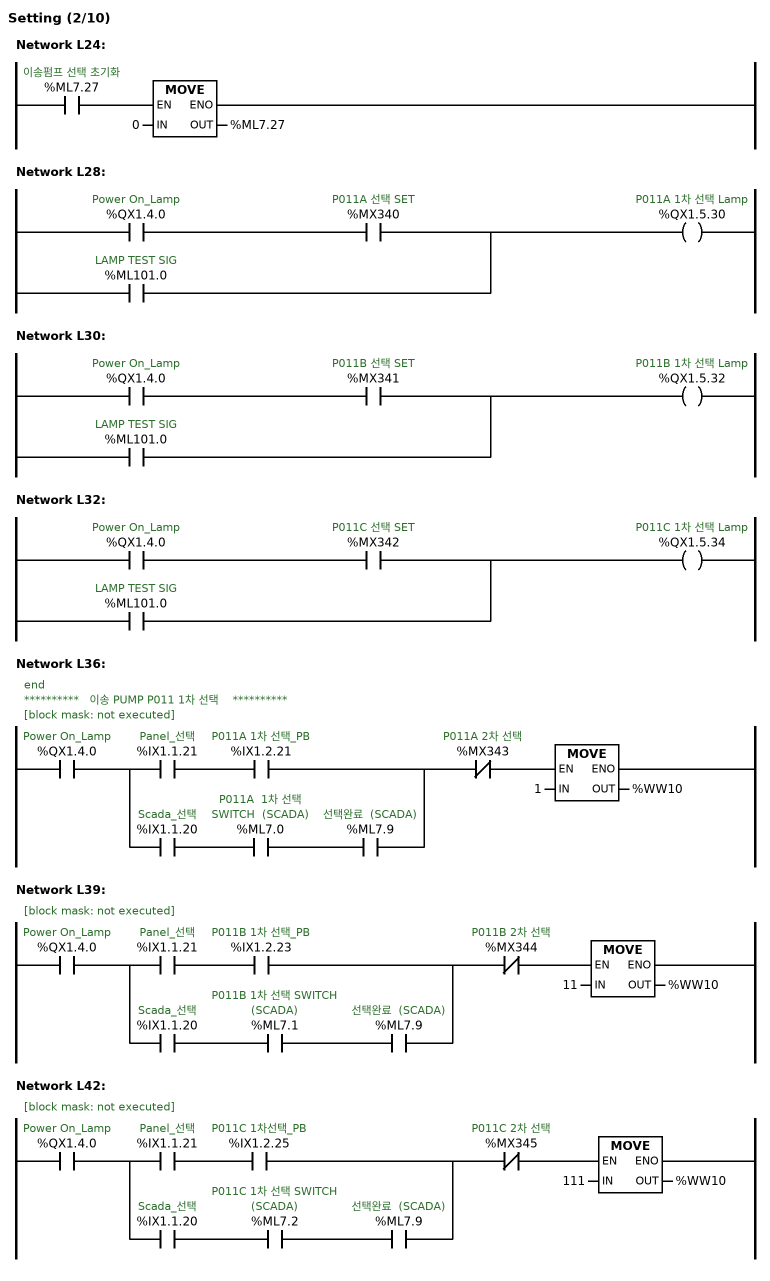
(* Rung L24 *)
IF %ML7.27 THEN %ML7.27 := 0; END_IF;
(*  *)
(* Rung L28 *)
%QX1.5.30 := (%QX1.4.0 AND %MX340) OR %ML101.0;
(* Rung L30 *)
%QX1.5.32 := (%QX1.4.0 AND %MX341) OR %ML101.0;
(* Rung L32 *)
%QX1.5.34 := (%QX1.4.0 AND %MX342) OR %ML101.0;
(* end *)
(* **********   이송 PUMP P011 1차 선택    ********** *)
(* Rung L36 is block-masked: not executed *)
// IF %QX1.4.0 AND ((%IX1.1.21 AND %IX1.2.21) OR (%IX1.1.20 AND %ML7.0 AND %ML7.9)) AND NOT %MX343 THEN
//     %WW10 := 1;
// END_IF;
(* Rung L39 is block-masked: not executed *)
// IF %QX1.4.0 AND ((%IX1.1.21 AND %IX1.2.23) OR (%IX1.1.20 AND %ML7.1 AND %ML7.9)) AND NOT %MX344 THEN
//     %WW10 := 11;
// END_IF;
(* Rung L42 is block-masked: not executed *)
// IF %QX1.4.0 AND ((%IX1.1.21 AND %IX1.2.25) OR (%IX1.1.20 AND %ML7.2 AND %ML7.9)) AND NOT %MX345 THEN
//     %WW10 := 111;
// END_IF;

